TEXTLIST stationLinked
  0 = 'Unlinked'
  1 = 'Linked'
   = ''
END_TEXTLIST

(* stored: Version 1.1.0.1, ProductVersion 3.1.4024.11
   TextList stationLinked: Id {bc776bb3-f58e-0305-1823-56f4a0009dd0} *)
